FUNCTION F_GetSBGaugeReadings : ST_SBGaugeReadings
VAR_INPUT
END_VAR
VAR
	stReadings : ST_SBGaugeReadings := (
		fDPPiraniVal:= GVL_BTS_VAC.fb_DP_GPI.PG.rPRESS,
		eDPPiraniState:= GVL_BTS_VAC.fb_DP_GPI.PG.eState,
		fDPColdCathodeVal:= GVL_BTS_VAC.fb_DP_GCC.IG.rPRESS,
		eDPColdCathodeState:= GVL_BTS_VAC.fb_DP_GCC.IG.eState,
		fPumpStationPirani1Val:= GVL_BTS_VAC.fb_PP_GPI_1.PG.rPRESS,
		ePumpStationPirani1State:= GVL_BTS_VAC.fb_PP_GPI_1.PG.eState,
		fPumpStationPirani2Val:= GVL_BTS_VAC.fb_PP_GPI_2.PG.rPRESS, 
		ePumpStationPirani2State:= GVL_BTS_VAC.fb_PP_GPI_2.PG.eState,
		fPumpStationColdCathodeVal:= GVL_BTS_VAC.fb_PP_GCC.IG.rPRESS,
		ePumpStationColdCathodeState:= GVL_BTS_VAC.fb_PP_GCC.IG.eState);
END_VAR

F_GetSBGaugeReadings := stReadings;

END_FUNCTION

(* stored: Version 1.1.0.1, ProductVersion 3.1.4024.0
   POU F_GetSBGaugeReadings: Id {87a652bb-93d8-46d8-bd90-4b26a57bdd2d}, SpecialFunc None *)
